// LS Electric XG5000 project: 0205 인버터통신
// PLC LSPLC

PROGRAM NewProgram (task: 스캔 프로그램)

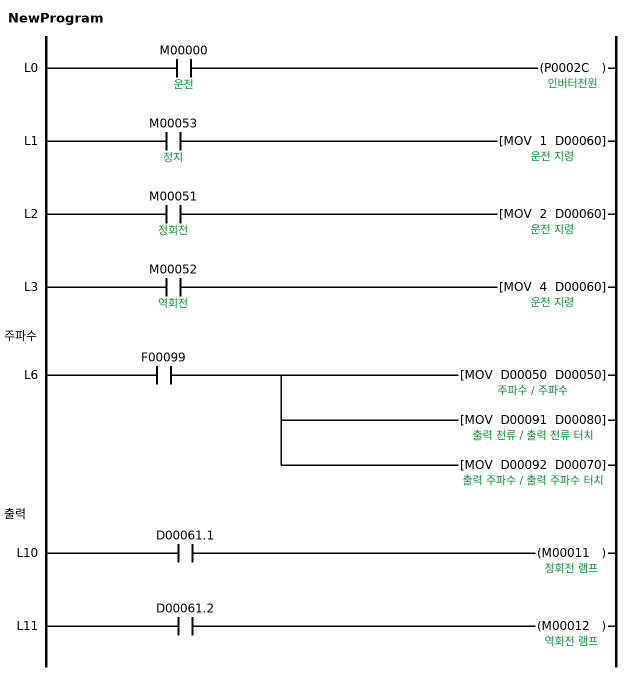
; L0
LOAD      M00000	// 운전
OUT       P0002C	// 인버터전원
; L1
LOAD      M00053	// 정지
MOV       1 D00060	// 운전 지령
; L2
LOAD      M00051	// 정회전
MOV       2 D00060	// 운전 지령
; L3
LOAD      M00052	// 역회전
MOV       4 D00060	// 운전 지령
주파수:
; L6
LOAD      F00099
MOV       D00050 D00050	// 주파수 / 주파수
MOV       D00091 D00080	// 출력 전류 / 출력 전류 터치
MOV       D00092 D00070	// 출력 주파수 / 출력 주파수 터치
출력:
; L10
LOAD      D00061.1
OUT       M00011	// 정회전 램프
; L11
LOAD      D00061.2
OUT       M00012	// 역회전 램프